(* Schneider Machine Expert - Basic project Bandeira_mastro, file version 2.7.0.0 *)
(* ProjectInformations: Name=Novo projeto *)

HARDWARE
  Cpu 0: TM221CE40R
  EthernetConfiguration: NetworkName=M221, IpAllocationMode=FixedAddress, IpAddress=0.0.0.0, SubnetMask=0.0.0.0
  SerialLineConfiguration: Baud=Baud19200, Parity=ParityEven, DataBits=DataBits8, StopBits=StopBits1, PhysicalMedium=PhysicalMediumRs485, TransmissionMode=TransmissionModeModbusRtu, SlaveId=1, Addressing=SlaveAddressing
  MastTask: UsePeriodScanMode=false, PeriodScan=100
  FastTask: Period=255
  CpuBehavior: StartingMode=StartAsPreviousState, AutoSaveRamOnEeprom=true, WatchdogPeriod=250

SYMBOLS  (address, symbol, comment, settings)
  %M0       PULSO  "Pulso"
  %M1       CT_PULSO  "Corta Pulso"
  %M2       P1  "Passo 1"
  %M3       P2  "Passo 2"
  %M4       P3  "Passo 3"
  %M5       P4  "Passo 4"
  %M6       PULSO_2  "Pulso 2"
  %M7       CT_PULSO_2  "Corta pulso 2"
  %M8       CT_PULSO_3  "Corta Pulso 3"
  %M9       PULSO_3  "Pulso 3"
  %I0.0     SA  "Sensor Alto"
  %I0.1     SB  "Sensor baixo"
  %I0.2     B0  "Botoeira Start"
  %I0.3     B1  "Botoeira UP"
  %I0.4     B2  "Botoeira Down"
  %Q0.0     RL0_UP  "Motor UP"
  %Q0.1     RL1_DW  "Motor Down"
  %Q0.2     L0  "Lampada Start"
  %Q0.3     L1  "Lampada UP"
  %Q0.4     L2  "Lampada Down"

POU Passos
  (* SectionNumber=1 *)

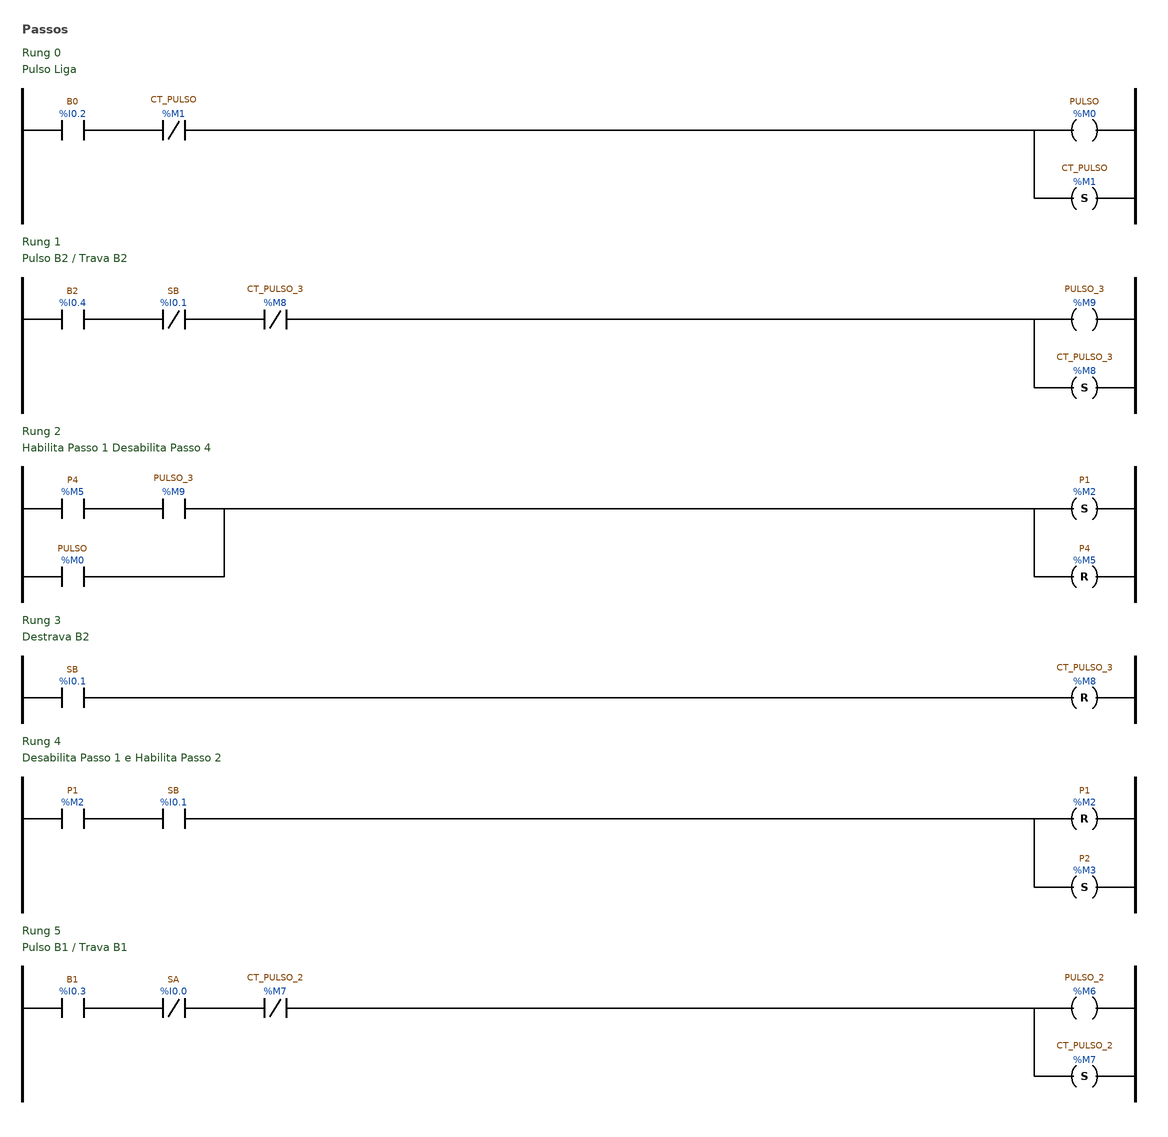

// Rung 0
// Pulso Liga
  LD %I0.2                (* B0 *)
  ANDN %M1                (* CT_PULSO *)
  ST %M0                  (* PULSO *)
  S %M1                   (* CT_PULSO *)
  // as ST:
  //   PULSO := B0 AND NOT CT_PULSO;
  //   IF B0 AND NOT CT_PULSO THEN CT_PULSO := TRUE; END_IF;

// Rung 1
// Pulso B2 / Trava B2
  LD %I0.4                (* B2 *)
  ANDN %I0.1              (* SB *)
  ANDN %M8                (* CT_PULSO_3 *)
  ST %M9                  (* PULSO_3 *)
  S %M8                   (* CT_PULSO_3 *)
  // as ST:
  //   PULSO_3 := B2 AND NOT SB AND NOT CT_PULSO_3;
  //   IF B2 AND NOT SB AND NOT CT_PULSO_3 THEN CT_PULSO_3 := TRUE; END_IF;

// Rung 2
// Habilita Passo 1 Desabilita Passo 4
  LD %M5                  (* P4 *)
  AND %M9                 (* PULSO_3 *)
  OR %M0                  (* PULSO *)
  S %M2                   (* P1 *)
  R %M5                   (* P4 *)
  // as ST:
  //   IF P4 AND PULSO_3 OR PULSO THEN P1 := TRUE; END_IF;
  //   IF P4 AND PULSO_3 OR PULSO THEN P4 := FALSE; END_IF;

// Rung 3
// Destrava B2
  LD %I0.1                (* SB *)
  R %M8                   (* CT_PULSO_3 *)
  // as ST:
  //   IF SB THEN CT_PULSO_3 := FALSE; END_IF;

// Rung 4
// Desabilita Passo 1 e Habilita Passo 2
  LD %M2                  (* P1 *)
  AND %I0.1               (* SB *)
  R %M2                   (* P1 *)
  S %M3                   (* P2 *)
  // as ST:
  //   _t1 := P1 AND SB;
  //   IF _t1 THEN P1 := FALSE; END_IF;
  //   IF _t1 THEN P2 := TRUE; END_IF;

// Rung 5
// Pulso B1 / Trava B1
  LD %I0.3                (* B1 *)
  ANDN %I0.0              (* SA *)
  ANDN %M7                (* CT_PULSO_2 *)
  ST %M6                  (* PULSO_2 *)
  S %M7                   (* CT_PULSO_2 *)
  // as ST:
  //   PULSO_2 := B1 AND NOT SA AND NOT CT_PULSO_2;
  //   IF B1 AND NOT SA AND NOT CT_PULSO_2 THEN CT_PULSO_2 := TRUE; END_IF;

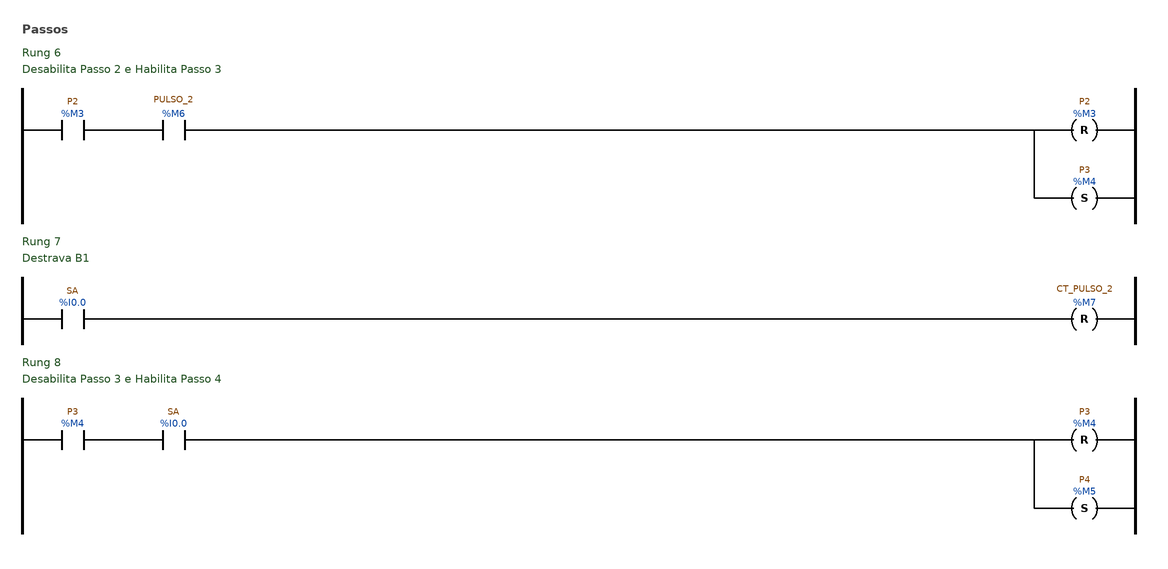

// Rung 6
// Desabilita Passo 2 e Habilita Passo 3
  LD %M3                  (* P2 *)
  AND %M6                 (* PULSO_2 *)
  R %M3                   (* P2 *)
  S %M4                   (* P3 *)
  // as ST:
  //   _t1 := P2 AND PULSO_2;
  //   IF _t1 THEN P2 := FALSE; END_IF;
  //   IF _t1 THEN P3 := TRUE; END_IF;

// Rung 7
// Destrava B1
  LD %I0.0                (* SA *)
  R %M7                   (* CT_PULSO_2 *)
  // as ST:
  //   IF SA THEN CT_PULSO_2 := FALSE; END_IF;

// Rung 8
// Desabilita Passo 3 e Habilita Passo 4
  LD %M4                  (* P3 *)
  AND %I0.0               (* SA *)
  R %M4                   (* P3 *)
  S %M5                   (* P4 *)
  // as ST:
  //   _t1 := P3 AND SA;
  //   IF _t1 THEN P3 := FALSE; END_IF;
  //   IF _t1 THEN P4 := TRUE; END_IF;

POU Sequencia
  (* SectionNumber=2 *)

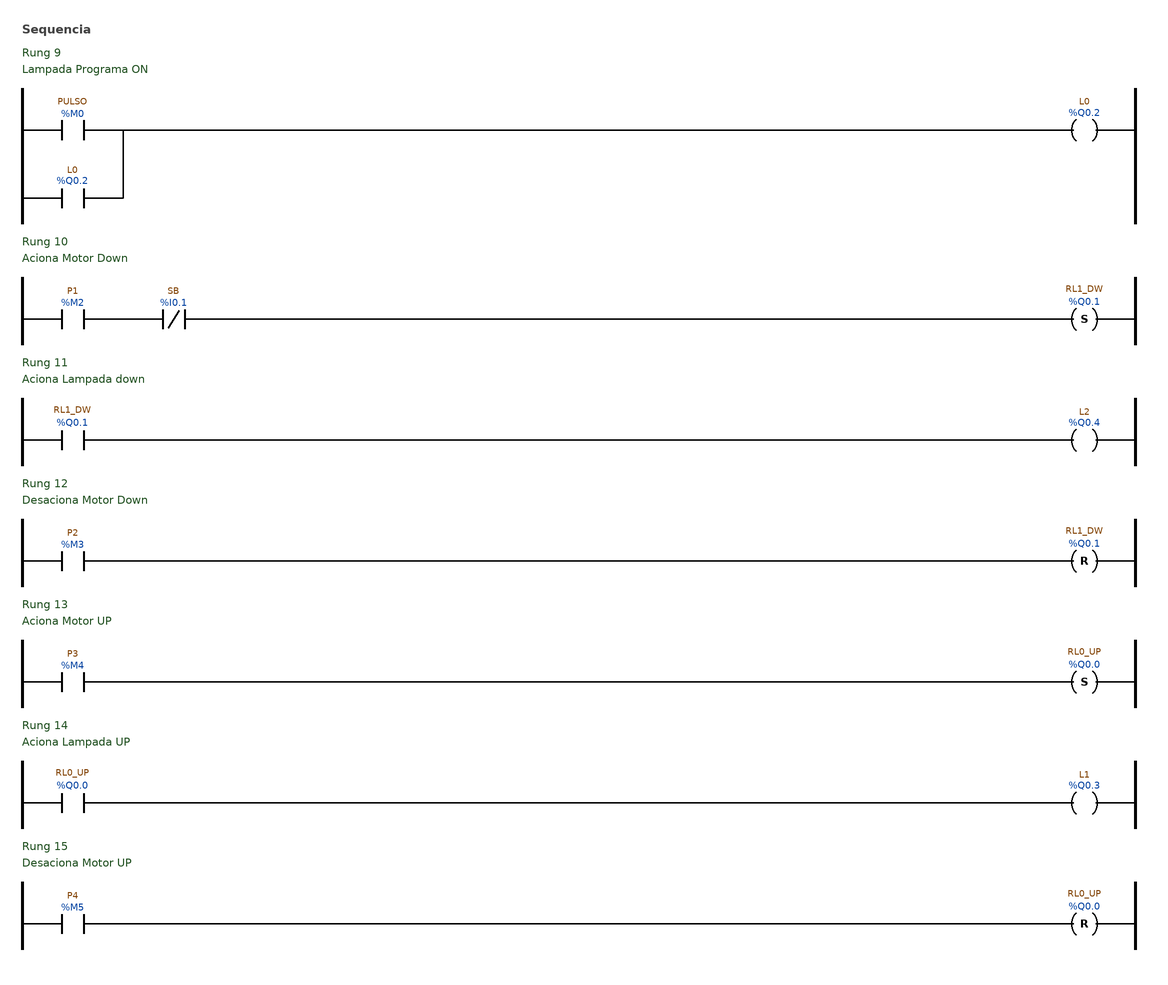

// Rung 9
// Lampada Programa ON
  LD %M0                  (* PULSO *)
  OR %Q0.2                (* L0 *)
  ST %Q0.2                (* L0 *)
  // as ST:
  //   L0 := PULSO OR L0;

// Rung 10
// Aciona Motor Down
  LD %M2                  (* P1 *)
  ANDN %I0.1              (* SB *)
  S %Q0.1                 (* RL1_DW *)
  // as ST:
  //   IF P1 AND NOT SB THEN RL1_DW := TRUE; END_IF;

// Rung 11
// Aciona Lampada down
  LD %Q0.1                (* RL1_DW *)
  ST %Q0.4                (* L2 *)
  // as ST:
  //   L2 := RL1_DW;

// Rung 12
// Desaciona Motor Down
  LD %M3                  (* P2 *)
  R %Q0.1                 (* RL1_DW *)
  // as ST:
  //   IF P2 THEN RL1_DW := FALSE; END_IF;

// Rung 13
// Aciona Motor UP
  LD %M4                  (* P3 *)
  S %Q0.0                 (* RL0_UP *)
  // as ST:
  //   IF P3 THEN RL0_UP := TRUE; END_IF;

// Rung 14
// Aciona Lampada UP
  LD %Q0.0                (* RL0_UP *)
  ST %Q0.3                (* L1 *)
  // as ST:
  //   L1 := RL0_UP;

// Rung 15
// Desaciona Motor UP
  LD %M5                  (* P4 *)
  R %Q0.0                 (* RL0_UP *)
  // as ST:
  //   IF P4 THEN RL0_UP := FALSE; END_IF;
